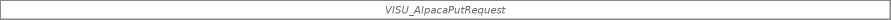
VISUALIZATION VISU_AlpacaPutNoArgs  // 891x20
VAR_IN_OUT
	stInstance : ST_AlpacaPutRequest;
END_VAR
    Frame (0,0 891x20)
        shows VISU_AlpacaPutRequest(stInstance := stInstance)
END_VISUALIZATION

(* stored: Version 1.1.0.1, ProductVersion 3.1.4024.12
   Visu VISU_AlpacaPutNoArgs: Id {0403a2cc-7ff0-44a8-b6f5-b5b2057be8d5} *)
